{attribute 'qualified_only'}
VAR_GLOBAL CONSTANT
	RISED		: Strings.Str := 'Rised';
	LOWERED		: Strings.Str := 'Lowered';
END_VAR

(* stored: Version 1.1.0.1
   GVL CFLAG: Id {7eeb824d-f799-4ea6-8deb-df670219d7f4} *)
